{attribute 'linkalways'} 
{attribute 'no_explicit_call' := 'This FB is a CLASS and must be accessed using methods or properties'}
{attribute 'enable_dynamic_creation'}
FUNCTION_BLOCK _ETcVnClusteringAlgorithm EXTENDS EnumDatatypeBase
VAR
	localData : ETcVnClusteringAlgorithm;
	activeData : REFERENCE TO ETcVnClusteringAlgorithm;
	enumBaseDatatype : _DINT(localData);
END_VAR

METHOD PRIVATE AddLocalEnumeration
VAR_INPUT
	Enumeration : T_MAXSTRING;
	Value : ETcVnClusteringAlgorithm;
END_VAR
AddEnumeration(Enumeration, Value);
END_METHOD

PROPERTY PUBLIC Address : PVOID
GET
Address := ADR(activeData);
END_GET
END_PROPERTY

METHOD PUBLIC ClearReference
VAR_INPUT
END_VAR
activeData REF= localData;
SetBaseDatatypeReference();
END_METHOD

METHOD PUBLIC Clone : I_Datatype
VAR
    pClone : POINTER TO _ETcVnClusteringAlgorithm;
END_VAR
pClone := __NEW(_ETcVnClusteringAlgorithm(InitialValue := Value));
Clone := pClone^;
END_METHOD

METHOD FB_init : BOOL
VAR_INPUT
	bInitRetains : BOOL; // if TRUE, the retain variables are initialized (warm start / cold start)
	bInCopyCode : BOOL;  // if TRUE, the instance afterwards gets moved into the copy code (online change)
	InitialValue : ETcVnClusteringAlgorithm;
END_VAR
localData := InitialValue;
AddBaseDatatype(enumBaseDatatype);
ClearReference();

AddLocalEnumeration('TCVN_CA_KMEANSPP', ETcVnClusteringAlgorithm.TCVN_CA_KMEANSPP);
AddLocalEnumeration('TCVN_CA_LBG', ETcVnClusteringAlgorithm.TCVN_CA_LBG);
END_METHOD

PROPERTY PUBLIC Identifier : T_MAXSTRING
GET
Identifier := 'ETcVnClusteringAlgorithm';
END_GET
END_PROPERTY

METHOD IsEnumeratorValueEqual : BOOL
VAR_INPUT
	Enumerator : I_KeyValueForwardEnumerator;
END_VAR
VAR
	storedValue : ETcVnClusteringAlgorithm;
END_VAR
IF NOT Enumerator.TryGet(storedValue) THEN
	RETURN;
END_IF

IsEnumeratorValueEqual := storedValue = activeData;
END_METHOD

METHOD PUBLIC MakeReferenceTo
VAR_INPUT
	ReferenceTarget : REFERENCE TO ETcVnCalibrationPatternOrigin;
END_VAR
activeData REF= ReferenceTarget;
SetBaseDatatypeReference();
END_METHOD

METHOD PROTECTED SetBaseDatatypeReference
VAR_INPUT
END_VAR
enumBaseDatatype.MakeReferenceTo(activeData);
END_METHOD

PROPERTY PUBLIC Size : UDINT
GET
Size := SIZEOF(activeData);
END_GET
END_PROPERTY

METHOD TryMakeReferenceTo : BOOL
VAR_INPUT
	Target : I_Datatype;
END_VAR
VAR
	targetAsEnum : I_EnumDatatype;
	pTargetData : POINTER TO ETcVnClusteringAlgorithm;
END_VAR
IF NOT Target.TryResolveAsEnumDatatype(targetAsEnum) THEN
	RETURN;
END_IF

IF targetAsEnum.Identifier <> Identifier THEN
	RETURN;
END_IF

pTargetData := Target.Address;
activeData REF= pTargetData^;
SetBaseDatatypeReference();
TryMakeReferenceTo := TRUE;
END_METHOD

PROPERTY PUBLIC Value : ETcVnClusteringAlgorithm
GET
Value := activeData;
END_GET
SET
activeData := Value;
END_SET
END_PROPERTY

END_FUNCTION_BLOCK

(* stored: Version 1.1.0.1
   POU _ETcVnClusteringAlgorithm: Id {9c6fb4e6-8044-0c70-13f7-f48618195223}, SpecialFunc None
   Folder Constructor: Id {9c538685-f722-07e5-1a95-68cbf9454740}
   Folder Private: Id {8f387a5e-313f-076a-03cc-c211aa214f7d}
   Folder Protected: Id {14483baf-61a8-0dd7-36ff-3a9b0318a718}
   Method AddLocalEnumeration: Id {67b76513-e5eb-0772-1b34-7da709a1df3b}
   Property Address: Id {32812d35-d5ce-0975-0346-08a724669b54}
   Get Get: Id {e9355d1c-dba1-0756-387a-a34d4fc374e3}
   Method ClearReference: Id {0aa735db-d62b-0847-1893-fd4d37273fee}
   Method Clone: Id {de1ef00a-7755-0b52-2763-36784b9c74eb}
   Method FB_init: Id {281361bc-d1e9-0828-348f-84e851d3d6aa}
   Property Identifier: Id {4672cc82-ec8a-004c-353d-e360642fe184}
   Get Get: Id {a0547ad5-3edc-0444-0029-574f8198093c}
   Method IsEnumeratorValueEqual: Id {a54fdbfe-1118-0cdf-220b-129e6515554f}
   Method MakeReferenceTo: Id {fbd5c6cc-0645-0b87-2971-75e92f7ba48b}
   Method SetBaseDatatypeReference: Id {710c7d16-003e-0010-390c-0db87efa3f99}
   Property Size: Id {014408c8-3013-05a2-2760-aead157faaf5}
   Get Get: Id {1db9b1fd-e96e-053b-2267-22ae6cab8144}
   Method TryMakeReferenceTo: Id {713adf2b-7667-0811-08d7-046049b291c2}
   Property Value: Id {8d423a1e-d01d-0a59-0056-73f3d73eb0f2}
   Get Get: Id {30336e6c-f767-0cd7-3bc4-cda222266b99}
   Set Set: Id {5c6a01bd-bc9b-094a-2cfb-70c496307d37} *)
